// TIA Portal V20 export
DATA_BLOCK "ComErrText"   // DB370
{ S7_Optimized_Access := 'TRUE' }
// stored: AutoNumber false, MemoryReserve 0
   VAR
      Plc : "TypeHeaderPlc";   // Header Plc
      Rd : Struct
         Pc : Struct
            watchdog : Bool;
            bit01 : Bool;
            bit02 : Bool;
            bit03 : Bool;
            bit04 : Bool;
            bit05 : Bool;
            bit06 : Bool;
            ack : Bool;
            word2 : Word;
            word4 : Word;
            word6 : Word;
            word8 : Word;
         END_STRUCT;
         language { S7_SetPoint := 'True'} : Array[1..3] of WString[2];   // language for alarm text [ISO639-1] (not used)
      END_STRUCT;
      Sd : Struct
         Pc : Struct
            watchdog : Bool;
            bit01 : Bool;
            bit02 : Bool;
            bit03 : Bool;
            bit04 : Bool;
            bit05 : Bool;
            bit06 : Bool;
            ack : Bool;
            word2 : Word;
            word4 : Word;
            word6 : Word;
            word8 : Word;
         END_STRUCT;
         language { S7_SetPoint := 'True'} : Array[1..3] of WString[2];   // language for alarm text [ISO639-1]
         errAct { ExternalAccessible := 'False'; ExternalVisible := 'False'; ExternalWritable := 'False'} : Array[1..20] of Struct   // alarm text for the most prior actual alarms on the plc
            idProd : UInt;   // producer Id (for Plc: 0=Program_Alarm, 4=SysDiag, 5=MotionControl, 6=Security, 8=GRAPH, 9=ProDiag)
            id : UInt;   // alarm Id (nr of alarm in the plc)
            prio : UInt;   // 0 .. 16 (0-1=info, 2=safety, 3=warning, 4-16=fault)
            timeStamp : LDT;   // UTC time [8Byte, LDT#2008-10-25-08:12:34.567]
            alarm : Array[1..3] of WString[254];   // alarm text
            info : Array[1..3] of WString[254];   // info text, cause of the alarm
            remedy : Array[1..3] of WString[254];   // remedy text, suggestion how to fix the fault
         END_STRUCT;
         errList : Struct   // alarm text to fill error list on Pc
            idProd : UInt;   // producer Id (for Plc: 0=Program_Alarm, 4=SysDiag, 5=MotionControl, 6=Security, 8=GRAPH, 9=ProDiag)
            id : UInt;   // alarm Id (Nr in error List)
            prio : UInt;   // 0 .. 16 (0-1=info, 2=safety, 3=warning, 4-16=fault)
            timeStamp : LDT;   // UTC time [8Byte, LDT#2008-10-25-08:12:34.567]
            alarm : Array[1..3] of WString[254];   // alarm text
            info : Array[1..3] of WString[254];   // info text, cause of the alarm
            remedy : Array[1..3] of WString[254];   // remedy text, suggestion how to fix the fault
         END_STRUCT;
      END_STRUCT;
   END_VAR
BEGIN
END_DATA_BLOCK
